{attribute 'linkalways'} 
{attribute 'no_explicit_call' := 'This FB is a CLASS and must be accessed using methods or properties'}
{attribute 'enable_dynamic_creation'}
FUNCTION_BLOCK FINAL MUL_REAL EXTENDS Node
VAR
	in1 : _REAL(0.0);
	in2 : _REAL(0.0);
	out : _REAL(0.0);
END_VAR

METHOD PUBLIC Clone : I_Node
VAR
	pNode : POINTER TO MUL_REAL;
END_VAR
pNode := __NEW(MUL_REAL);
Clone := pNode^;
END_METHOD

METHOD FB_init : BOOL
VAR_INPUT
	bInitRetains : BOOL; // if TRUE, the retain variables are initialized (warm start / cold start)
	bInCopyCode : BOOL;  // if TRUE, the instance afterwards gets moved into the copy code (online change)
END_VAR
AddInput('in1',THIS^.in1);
AddInput('in2',THIS^.in2);
AddOutput('out', THIS^.out);
END_METHOD

METHOD PROTECTED OnExecute
VAR
END_VAR
out.Value := in1.Value * in2.Value;
END_METHOD

END_FUNCTION_BLOCK

(* stored: Version 1.1.0.1, ProductVersion 3.1.4024.15
   POU MUL_REAL: Id {cb49e716-6761-4d17-bee6-1a87db87de55}, SpecialFunc None
   Folder Constructor: Id {5361ab84-fb74-4e10-acbd-e9ae1794a17c}
   Method Clone: Id {a27317bd-f5a8-4d01-b612-e9a21a8a2b76}
   Method FB_init: Id {5bf7ade2-d327-4176-bd8c-cd5b3057b126}
   Method OnExecute: Id {5f622b3a-feb0-45b3-99e7-512d2145d9b5} *)
